Omron CX-Programmer project NewProject (CX-Programmer 9.03)

# PLC NewPLC1: CP1L L
; plc-pompa

## Global symbols (name address type ; comment)
0.00 BOOL  ; STOP
0.01 BOOL  ; START
1.00 BOOL  ; lampu

## Program NewProgram1 (cyclic task 0)

### Section Section1

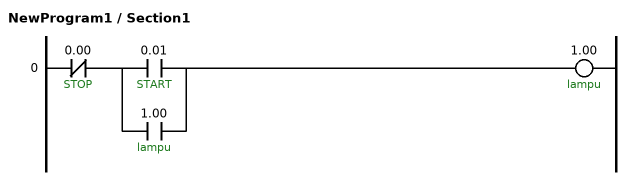
; rung 0
LDNOT 0.00  ; STOP
LD 0.01  ; START
OR 1.00  ; lampu
ANDLD
OUT 1.00  ; lampu

### Section END
; rung 0
END(001)